INTERFACE I_NullEntry EXTENDS I_FileSystemEntry

END_INTERFACE

(* stored: Version 1.1.0.1, ProductVersion 3.1.4024.9
   Itf I_NullEntry: Id {183f6e87-ae3c-49de-97ef-7d2b9df21cdd} *)
